FUNCTION_BLOCK SUBL_1_OK (* 2-variable data subscriber *)
  (* Standard: 61499-2 *)
  (* Version 1.0, 21-03-12, GASR, Universidade do Estado de Santa Catarina *)
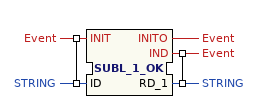
  EVENT_INPUT
    INIT WITH ID; (* Service initiaization *)
  END_EVENT
  EVENT_OUTPUT
    INITO; (* Initialization confirm *)
    IND WITH RD_1; (* Service indication *)
  END_EVENT
  VAR_INPUT
    ID : STRING; (* Default id is the FB instance name *)
  END_VAR
  VAR_OUTPUT
    RD_1 : STRING;
  END_VAR
  SERVICE PUBL_1_OK/SUBL_1_OK (* Data publication service *)
    SEQUENCE normal_establishment
      PUBL_1_OK.INIT(ID) -> PUBL_1_OK.INITO();
      SUBL_1_OK.INIT(ID) -> SUBL_1_OK.INITO();
    END_SEQUENCE
    SEQUENCE normal_data_transfer
      PUBL_1_OK.REQ(SD_1) -> Subl_1_OK.IND(RD_1);
    END_SEQUENCE
  END_SERVICE
END_FUNCTION_BLOCK
